{attribute 'enable_dynamic_creation'}
FUNCTION_BLOCK FutureMCMoveVelocity EXTENDS FB_AbstructFuture
VAR_INPUT
END_VAR
VAR_OUTPUT
END_VAR
VAR
	_fb_move_velo	: MC_MoveVelocity;
	_executor		: FB_Executor;
	_axis: REFERENCE TO AXIS_REF;
	_velocity : MC_LREAL;
	_direction : MC_DIRECTION;
	_acceleration: MC_LREAL;
	_deceleration: MC_LREAL;
	_jerk		: MC_LREAL;
	_option : ST_MoveOptions;
	_buffer_mode : MC_BufferMode ;
	_error_id :UDINT;
	_exec_state : UDINT;
	_abort_state : UINT;
END_VAR

METHOD abort : BOOL // Return TRUE if finish.
VAR_INST
	future_halt : FutureMcHalt;
END_VAR
CASE _abort_state OF
	0:
		_exec_state := 0;
		future_halt.set_parameters(_axis, _deceleration, _jerk);
		future_halt.future_name := 'HALT MOVE_RELATIVE';
		_executor.future := future_halt;
		_abort_state := 1;
	1:
		IF _executor.execute() AND _executor.nErrorID = 0 THEN
			_abort_state := 2;
		END_IF
		
		IF _executor.current_state = E_FutureExecutionState.wait_for_process THEN
			_executor.start();
		END_IF
	2:
		abort := TRUE;
END_CASE
END_METHOD

METHOD execute : BOOL // Return TRUE if finish.

CASE _exec_state OF
	0:
		_abort_state := 0;
		_fb_move_velo(Axis := _axis,Execute := FALSE);
		_fb_move_velo(
			Execute := TRUE,
			Axis := _axis,
			Direction := _direction,
			Velocity := _velocity,
			Acceleration := _acceleration,
			Deceleration := _deceleration,
			Jerk := _jerk,
			BufferMode := _buffer_mode,
			Options := _option
		);
		_exec_state := 1;
	1:
		IF _fb_move_velo.Busy THEN
			_fb_move_velo(Axis := _axis,Execute := FALSE);
		END_IF
END_CASE

_error_id := _fb_move_velo.ErrorID;
execute := _fb_move_velo.InVelocity OR _fb_move_velo.Error;
END_METHOD

METHOD init : BOOL // Return TRUE if finish.

VAR
	axis: INT;
END_VAR
_exec_state := 0;
_abort_state := 0;
_error_id := _fb_move_velo.ErrorID;
init := TRUE;
END_METHOD

PROPERTY nErrorID : UDINT
GET
nErrorID := _error_id;
END_GET
SET
END_SET
END_PROPERTY

METHOD set_options : BOOL
VAR_INPUT
	option : ST_MoveOptions;
END_VAR
_option := option;
END_METHOD

METHOD set_parameters : BOOL
VAR_INPUT
	axis : REFERENCE TO AXIS_REF;
	direction : MC_DIRECTION;
	velocity : MC_LREAL;
	acceleration	: MC_LREAL;		// Set deceleration in case let moving axis halt.
	deceleration	: MC_LREAL;		// Set deceleration in case let moving axis halt.
	jerk			: MC_LREAL;		// Set jerk in case let moving axis halt.
	buffer_mode : MC_BufferMode;
END_VAR
_axis REF= axis;
_velocity := velocity;
_direction := direction;
_acceleration := acceleration;
_deceleration := deceleration;
_jerk := jerk;
_buffer_mode := buffer_mode;
END_METHOD

END_FUNCTION_BLOCK

(* stored: Version 1.1.0.1, ProductVersion 3.1.4024.12
   POU FutureMCMoveVelocity: Id {29148965-5e10-4a14-94be-705867904fbe}, SpecialFunc None
   Method abort: Id {72fcad41-759f-41d6-bfdc-0ea86e66e7a3}
   Method execute: Id {199850b7-b50d-4a98-900c-cfddcfc3c30c}
   Method init: Id {95bb8aca-b748-477b-ae1d-3c5d6d817a51}
   Property nErrorID: Id {d0c28b4c-d1ff-4af5-bd15-853506ce923b}
   Get Get: Id {c772ce53-a26d-4703-bf4d-5dec352edf66}
   Set Set: Id {507adb7d-f7fc-426b-a973-6b7526503bdd}
   Method set_options: Id {bf17cdaf-530f-4c56-93b8-8584092489c0}
   Method set_parameters: Id {49a5db17-1b30-4653-ab84-e6b95faefca6} *)
